// TIA Portal V19 export
TYPE "Prod_Mode"
   STRUCT
      MES_ON : Bool;   // inserimento ordini da MES è Acceso
      Cambio_Ordine_Automatico : Bool;   // Cambio automatico dell'ordine di profuzione è Acceso
   END_STRUCT;
END_TYPE
